Staubli VAL3: onF2Event.pgx

program onF2Event()
  local string l_sMessage
  local string l_sEvent
  local string l_sFilter
  local num l_nIndex
  local num i
begin
//  // look if the bButton is enable
//  if bButton[1]
//    //
//    // make a selection list
//    //
//    // 0) Filter by name
//    //
//    call use:clear(0,13)
//    call use:type(5,13,sMenu[1])
//    call language:message(l_sMessage,85)
//    call use:timerDialog(l_sMessage+": ",0)
//    l_sFilter=saveData:sTrajFilter
//    call use:read(20+(len(l_sMessage)/2)+1,5,l_sFilter,10,false)
//    if !use:bUseEscape
//      saveData:sTrajFilter=l_sFilter
//    endIf

//    // update
//    call buildList()
//    use:bUseRefresh=true
//    // release the key
//    call use:nullKey(nKey)
//  endIf
end
